FUNCTION F_Temperature : REAL
VAR_INPUT
	Input																: INT;
	Offset																: REAL;
END_VAR
VAR
END_VAR

// F_Temperature
// Rev 1.0 - December 28, 2023

F_Temperature															:= INT_TO_REAL(Input) / 10.0 + Offset;

END_FUNCTION

(* stored: Version 1.1.0.1, ProductVersion 3.1.4024.12
   POU F_Temperature: Id {884ae771-b46f-4b70-94ce-bbcbd3306258}, SpecialFunc None *)
